// TIA Portal V20 export
TYPE "UDT_RFID_Basic_Data"
   STRUCT
      Pallet_ID : Int;   // 托盘号
      Repair_Status : Int;   // 返修标致（0：无状态，1：正常件，2：返修件）
      Reserves_1 : Int;   // 预留
      Reserves_2 : Int;   // 预留
      Reserves_3 : Int;   // 预留
      Reserves_4 : Int;   // 预留
      Reject_Stn_Number : String[8];   // 拒绝工位（由不合格工位写入）
      UpLoad_Stn_Number : String[8];   // 上线工位（返修上线工位写入）
      Reserves_5 : Int;   // 预留
      PLCProductWorkOrderID : String[66];   // 产品工单号数据
      PLCProductModelID : String[32];   // 产品型号信息
      PLCProductRecipeID : Word;   // 产品配方号数据
      PLCProductSN : String[96];   // 产品序列号
      PLCProductPN : String[96];   // 产品批次号
      PLCCurrentProductSN : String[96];   // 当前处理的产品序列号
      PLCProductCustomerSN : String[96];   // 产品客户序列号
      PLCProductCustomerSNType : Word;   // 产品客户序列号类型
      Reserves_6 : Int;   // 预留
      Reserves_7 : Int;   // 预留
      Reserves_8 : Int;   // 预留
      Reserves_9 : Int;   // 预留
   END_STRUCT;
END_TYPE
